{attribute 'GeneratedUsingTerminal: EK1122-0000-0018'}
{attribute addProperty BoxType "EK1122-0000-0018"}
{attribute addProperty Id "Beckhoff_EPP6xxxsub_EK1100EK1100_1FC0878B2A_0001_EPP6001_0002_0016EPP6001_B53D58EE52A_0002_EPP6001_0002_0017EPP6001_B53D58EE52A_0003_EPP6001_0002_0018EPP6001_B53D58EE52A_0004_EPP6002_0002_0016EPP6002_E77396C2100A_0005_EPP6002_0002_0017EPP6002_E77396C2100A_0006_EPP6002_0002_0018EPP6002_A97F2B25100A_0007_EPP6002_0002_0019EPP6002_A97F2B25100A_0008_EPP6090_0000_0017EPP6090_9BC1C0C414A_0009_EPP6228_0022_0016EPP6228_5FAAB3C122"}
{attribute addProperty CRC "2891831584"}
{attribute addProperty Size "594"}
TYPE Beckhoff_EPP6xxxEK1122_AC5DD920 EXTENDS EK1122_1FC0878B :
STRUCT
	{attribute addProperty Name "Beckhoff_EPP6xxxsub_EK1100"}
	{attribute addProperty PreviousPort "Beckhoff EPP6xxxEK1122 : D"}
	Beckhoff_EPP6xxxsub_EK1100 : EK1100_1FC0878B;
	{attribute addProperty Name "A_0001_EPP6001_0002_0016"}
	{attribute addProperty PreviousPort "Beckhoff EPP6xxxsub EK1100 : C"}
	A_0001_EPP6001_0002_0016 : EPP6001_B53D58EE;
	{attribute addProperty Name "A_0002_EPP6001_0002_0017"}
	{attribute addProperty PreviousPort "A_0001(EPP6001-0002-0016) : B"}
	A_0002_EPP6001_0002_0017 : EPP6001_B53D58EE;
	{attribute addProperty Name "A_0003_EPP6001_0002_0018"}
	{attribute addProperty PreviousPort "A_0002(EPP6001-0002-0017) : B"}
	A_0003_EPP6001_0002_0018 : EPP6001_B53D58EE;
	{attribute addProperty Name "A_0004_EPP6002_0002_0016"}
	{attribute addProperty PreviousPort "A_0003(EPP6001-0002-0018) : B"}
	A_0004_EPP6002_0002_0016 : EPP6002_E77396C2;
	{attribute addProperty Name "A_0005_EPP6002_0002_0017"}
	{attribute addProperty PreviousPort "A_0004(EPP6002-0002-0016) : B"}
	A_0005_EPP6002_0002_0017 : EPP6002_E77396C2;
	{attribute addProperty Name "A_0006_EPP6002_0002_0018"}
	{attribute addProperty PreviousPort "A_0005(EPP6002-0002-0017) : B"}
	A_0006_EPP6002_0002_0018 : EPP6002_A97F2B25;
	{attribute addProperty Name "A_0007_EPP6002_0002_0019"}
	{attribute addProperty PreviousPort "A_0006(EPP6002-0002-0018) : B"}
	A_0007_EPP6002_0002_0019 : EPP6002_A97F2B25;
	{attribute addProperty Name "A_0008_EPP6090_0000_0017"}
	{attribute addProperty PreviousPort "A_0007(EPP6002-0002-0019) : B"}
	A_0008_EPP6090_0000_0017 : EPP6090_9BC1C0C4;
	{attribute addProperty Name "A_0009_EPP6228_0022_0016"}
	{attribute addProperty PreviousPort "A_0008(EPP6090-0000-0017) : B"}
	A_0009_EPP6228_0022_0016 : EPP6228_5FAAB3C1;
END_STRUCT
END_TYPE

(* stored: Version 1.2.0.0, ProductVersion 3.1.4024.9
   DUT Beckhoff_EPP6xxxEK1122_AC5DD920: Id {100f31b9-a3a1-453d-8ffd-4c25fac88f49} *)
